FUNCTION_BLOCK FB_RTUMaster_PcCOm_K EXTENDS FB_ModbusMaster_PcCOM
VAR_INPUT
	psKey : POINTER TO STRING(31);
END_VAR
VAR
	{attribute 'hide'}
	fbREEPROM_CFirmKey : FB_Cx7_Read_EEPROM_CFIRM_KEY;
END_VAR

SUPER^();
fbREEPROM_CFirmKey(psKey := psKey);

METHOD Run : BOOL /// call from FB_modbus
IF fbREEPROM_CFirmKey.bCorrectKey THEN
	iStepGeneral := E_ModBusMasterState.Running;
END_IF
Run := iStepGeneral=E_ModBusMasterState.Running;
END_METHOD

END_FUNCTION_BLOCK

(* stored: Version 1.1.0.1, ProductVersion 3.1.4024.12
   POU FB_RTUMaster_PcCOm_K: Id {58ed53c6-3323-47b3-91b0-8b163e376fa8}, SpecialFunc None
   Method Run: Id {4bad4141-abfe-4551-afca-10ae8c392ed2} *)
